PROGRAM DALI_COMM
VAR
	commLL		: ARRAY[1..GVL_IO.maxLLBus] OF Tc3_DALI.FB_KL6821Communication;
	
	commT1		: ARRAY[1..GVL_IO.maxT1Bus] OF Tc3_DALI.FB_KL6821Communication;
	commT2		: ARRAY[1..GVL_IO.maxT2Bus] OF Tc3_DALI.FB_KL6821Communication;
	commT3		: ARRAY[1..GVL_IO.maxT3Bus] OF Tc3_DALI.FB_KL6821Communication;
	commT4		: ARRAY[1..GVL_IO.maxT4Bus] OF Tc3_DALI.FB_KL6821Communication;
	commLS		: Tc3_DALI.FB_KL6821Communication;
	
	i : INT;
END_VAR
VAR CONSTANT
	
END_VAR

FOR i := 1 TO GVL_Variant.numLLBus DO
	commLL[i](
		stInData	:= GVL_IO.kl6821_LL_in[i],
		stOutData	:= GVL_IO.kl6821_LL_out[i],
	);
END_FOR

FOR i := 1 TO GVL_Variant.numT1Bus DO
	commT1[i](
		stInData	:= GVL_IO.kl6821_T1_in[i],
		stOutData	:= GVL_IO.kl6821_T1_out[i]
	);
END_FOR

FOR i := 1 TO GVL_Variant.numT2Bus DO
	commT2[i](
		stInData	:= GVL_IO.kl6821_T2_in[i],
		stOutData	:= GVL_IO.kl6821_T2_out[i]
	);
END_FOR

FOR i := 1 TO GVL_Variant.numT3Bus DO
	commT3[i](
		stInData	:= GVL_IO.kl6821_T3_in[i],
		stOutData	:= GVL_IO.kl6821_T3_out[i]
	);
END_FOR

FOR i := 1 TO GVL_Variant.numT4Bus DO
	commT4[i](
		stInData	:= GVL_IO.kl6821_T4_in[i],
		stOutData	:= GVL_IO.kl6821_T4_out[i]
	);
END_FOR

IF GVL_Variant.hasLSBus THEN
	commLS(
		stInData	:= GVL_IO.kl6821_LS_in,
		stOutData	:= GVL_IO.kl6821_LS_out
	);
END_IF

END_PROGRAM

(* stored: Version 1.1.0.1, ProductVersion 3.1.4024.11
   POU DALI_COMM: Id {5ac38050-9b14-4875-9d9e-9070976fdbca}, SpecialFunc None *)
